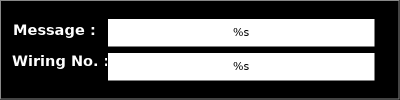
VISUALIZATION PUDetail  // 400x100
    Rectangle (0,0 400x100)
        OnMouseClick: CloseDialog Dialog=PUDetail, Result=None, NumpadKeypadSet=True
    Label (10,15 84x30), "Message :"
    Label (9,46 84x30), "Wiring No. :"
    Label (101,17 61x30)
    RoundedRectangle (107,18 268x29), "%s", tooltip "%s", text variable: HMI_GVL.sMessageError
        p4168582468: HMI_GVL.sMessageError
    RoundedRectangle (107,52 268x29), "%s", tooltip "%s", text variable: HMI_GVL.sWiringNo
        p4168582468: HMI_GVL.sWiringNo
END_VISUALIZATION

(* stored: Version 1.1.0.1, ProductVersion 3.1.4024.12
   Visu PUDetail: Id {087189a1-9876-4ab9-bc3b-9424227268bb} *)
